PROGRAM PRG_TEST
VAR
	fbExtractAnyStringTests			: FB_ExtractAnyStringTests;
	fbExtractStringTests			: FB_ExtratcStringTests;
	fbReplaceLongStringCharTests	: FB_ReplaceLongStringCharTests;
	fbLogHandlerTests				: FB_LogHandlerTests;
	
	fbValidateContentTests			: FB_CASE_ValidateContentTests;
END_VAR

//===================================================
//UNIT TEST EXECUTION

TcUnit.RUN();

//===================================================
//MANUAL TEST EXECUTION

PRG_ExtractAnyStringManual();
PRG_ExtractStringManual();
PRG_ReplaceLongSingleCharManual();
PRG_LogHandlerManual();

END_PROGRAM

(* stored: Version 1.1.0.1
   POU PRG_TEST: Id {08b43075-4f43-43da-b21b-f4c6343654c9}, SpecialFunc None *)
